// TIA Portal V20 export
TYPE "LER_typeRadiusMeasureMonitioing"
// stored: Access Published
   STRUCT
      Radius : LReal;
      Diameter : LReal;
   END_STRUCT;
END_TYPE
